FUNCTION F_DateTimeAsString_ms : T_MaxString
VAR_INPUT
    TimeStruct : TIMESTRUCT;
END_VAR
VAR
	FB_FormatString1 : FB_FormatString;
END_VAR

F_DateTimeAsString_ms := F_FormatStringEx2(
                             Format := '%s %s',
                             arg1   := F_TimeAsString_ms(TimeStruct),
                             arg2   := F_DateAsString(TimeStruct));

END_FUNCTION

(* stored: Version 1.1.0.1, ProductVersion 3.1.4024.3
   POU F_DateTimeAsString_ms: Id {792ea374-7462-0806-26f6-cb6adaaa325e}, SpecialFunc None *)
